// TIA Portal V20 export
TYPE "UDT_Service_ProcedureRawDataMedium"
   STRUCT
      procedure { S7_SetPoint := 'True'} : Array[0..15] of "UDT_MTP_ProcedureExtended";
   END_STRUCT;
END_TYPE
